Yaskawa INFORM job: COMARC_TEST_PACHWINA.JBI

/JOB
//NAME COMARC_TEST_PACHWINA
//POS
///NPOS 4,4,0,0,0,0
///TOOL 0
///POSTYPE ROBOT
///RECTAN
///RCONF 1,0,0,0,0,0,0,0,0,0,0,0,0,0,0,0,0,0,0,0,0,0,0,0
C00000=375.253,-82.900,-948.609,-0.0018,45.0017,-0.0064
C00001=392.031,136.513,-943.065,-0.0034,45.0030,-0.0075
C00002=375.256,-82.901,-955.880,-0.0026,45.0011,-0.0079
C00003=382.436,178.926,-955.867,-0.0033,45.0026,-0.0102
///RCONF 0,0,0,0,0,0,0,0,0,0,0,0,0,0,0,0,0,0,0,0,0,0,0,0
BC00000=3036.073
BC00001=3036.073
BC00002=3036.073
BC00003=3036.073
//INST
///DATE 2024/10/23 15:29
///ATTR SC,RW,RJ
////FRAME ROBOT
///GROUP1 RB1,BS1
NOP
REFP 1 C00000 BC00000
REFP 2 C00001 BC00001
MACRO1 MJ#(0) ARGF50
MOVL C00002 BC00002 V=16.7 PL=0
ARCON
COMARCON AMP=0.5 FREQ=2.5 ANGL=45.0 U/D=4800 L/R=3.0
MOVL C00003 BC00003 V=8.3
ARCOF
COMARCOF
END
